(* Logix 5000 project; controller batter_comorfords vendor 1 type 14 code 222 rev 33.11; software revision 33.00 *)

TASK MainTask (continuous, watchdog 500 ms) : MainProgram
TASK SafetyTask (periodic, rate 20 ms, priority 10, watchdog 20 ms, safety) : SafetyProgram

MODULES
   Local : vendor 1 type 14 code 222 (5069 0, rev 33.11)
      PF525_Stirrer : PowerFlex 525-EENET (Ethernet 192.168.2.13, rev 5.2, Output RPI 20 ms)   // 0.75KW
      PF525_FeedingPump_2 : PowerFlex 525-EENET (Ethernet 192.168.2.15, rev 5.2, Output RPI 20 ms)   // 0.75 kW
      PF525_FeedingPump_1 : PowerFlex 525-EENET (Ethernet 192.168.2.14, rev 5.2, Output RPI 20 ms)   // 0.75 KW
      Manifold_with_color : 2198-H008-ERS2 (Ethernet 192.168.2.17, rev 7.1, DSafety_Input RPI 10 ms, CSafety_Output RPI 20 ms, AMotionDiagnostics RPI 1 ms)
      Manifold_without_color : 2198-H008-ERS2 (Ethernet 192.168.2.18, rev 7.1, AMotionDiagnostics RPI 1 ms, DSafety_Input RPI 10 ms, CSafety_Output RPI 20 ms)
      X_axis : 2198-H008-ERS2 (Ethernet 192.168.2.19, rev 7.1, AMotionDiagnostics RPI 1 ms, CSafety_Output RPI 20 ms, DSafety_Input RPI 10 ms)
      Y_axis : 2198-H008-ERS2 (Ethernet 192.168.2.20, rev 7.1, AMotionDiagnostics RPI 1 ms, CSafety_Output RPI 20 ms, DSafety_Input RPI 10 ms)
      Z_axis : 2198-H008-ERS2 (Ethernet 192.168.2.21, rev 7.1, AMotionDiagnostics RPI 1 ms, CSafety_Output RPI 20 ms, DSafety_Input RPI 10 ms)
      U1_MCC1_IO : 1734-AENTR (Ethernet 192.168.2.12, rev 6.1, Output RPI 20 ms)
         U1_MCC1_DIG_In_1 : 1734-IB8 (PointIO 3, rev 3.1)
         U1_MCC1_DIG_In_2 : 1734-IB8 (PointIO 4, rev 3.1)
         U1_MCC1_DIG_In_3 : 1734-IB8 (PointIO 5, rev 3.1)
         U1_MCC1_ANA_In_1 : vendor 1 type 115 code 210 (PointIO 6, rev 3.1, Input RPI 80 ms)
         U1_MCC1_DIG_Out_1 : vendor 1 type 7 code 231 (PointIO 7, rev 3.1)
         U1_MCC1_DIG_Out_2 : 1734-OB8 (PointIO 8, rev 3.1)
         U1_MCC1_DIG_Out_3 : 1734-OB8 (PointIO 9, rev 3.1)
         U1_MCC1_DIG_Out_4 : 1734-OB8 (PointIO 10, rev 3.1)
         U1_MCC1_ANA_Out_1 : 1734-OE2C (PointIO 11, rev 3.1, Output RPI 80 ms)
         U1_MCC1_Safety_DIG_In_1 : vendor 1 type 35 code 15 (PointIO 1, rev 2.1, Input RPI 10 ms, Output RPI 20 ms)
         U1_MCC1_Safety_DIG_Out_1 : vendor 1 type 35 code 16 (PointIO 2, rev 2.1, Input RPI 10 ms, Output RPI 20 ms)
      U4_MCC1_IO : 1734-AENTR (Ethernet 192.168.2.16, rev 6.1, Output RPI 20 ms)
         U4_MCC1_DIG_In_1 : 1734-IB8 (PointIO 3, rev 3.1)
         U4_MCC1_DIG_In_2 : 1734-IB8 (PointIO 4, rev 3.1)
         U4_MCC1_DIG_In_3 : 1734-IB8 (PointIO 5, rev 3.1)
         U4_MCC1_ANA_In_1 : 1734-IE4C (PointIO 6, rev 3.1, Input RPI 80 ms)
         U4_MCC1_ANA_In_2 : 1734-IE4C (PointIO 7, rev 3.1, Input RPI 80 ms)
         U4_MCC1_DIG_Out_1 : vendor 1 type 7 code 231 (PointIO 8, rev 3.1)
         U4_MCC1_DIG_Out_2 : vendor 1 type 7 code 231 (PointIO 9, rev 3.1)
         U4_MCC1_DIG_Out_3 : vendor 1 type 7 code 231 (PointIO 10, rev 3.1)
         U4_MCC1_ANA_Out_1 : 1734-OE2C (PointIO 11, rev 3.1, Output RPI 80 ms)
         U4_MCC1_Safety_DIG_In_1 : vendor 1 type 35 code 15 (PointIO 1, rev 2.1, Input RPI 10 ms, Output RPI 20 ms)
         U4_MCC1_Safety_DIG_Out_1 : vendor 1 type 35 code 16 (PointIO 2, rev 2.1, Input RPI 10 ms, Output RPI 20 ms)
END_MODULES

VAR_GLOBAL   (* controller tags *)
   IA_1_1_LT01 : ALIAS FOR U1_MCC1_IO:6:I.Ch0Data;   // Level buffertank
   IA_1_1_PT01 : ALIAS FOR U1_MCC1_IO:6:I.Ch1Data;   // Pressure feeding pump 1
   IA_1_2_LT01 : ALIAS FOR U1_MCC1_IO:6:I.Ch3Data;   // Level buffertank
   IA_1_2_PT01 : ALIAS FOR U1_MCC1_IO:6:I.Ch2Data;   // Pressure color injection
   IA_4_1_PT01 : ALIAS FOR U4_MCC1_IO:6:I.Ch1Data;   // Pressure manifold color
   IA_4_1_PT02 : ALIAS FOR U4_MCC1_IO:6:I.Ch3Data;   // Pressure manifold no color
   IA_4_1_TT01 : ALIAS FOR U4_MCC1_IO:6:I.Ch0Data;   // Temperature manifold color
   IA_4_1_TT02 : ALIAS FOR U4_MCC1_IO:6:I.Ch2Data;   // Temperature manifold no color
   ID_1_1_CIP_FAULT : ALIAS FOR U1_MCC1_IO:4:I.5;   // Fault CIP pump soft starter
   ID_1_1_GS01_1 : ALIAS FOR U1_MCC1_IO:3:I.5;   // Guard switch 1.1
   ID_1_1_GS01_2 : ALIAS FOR U1_MCC1_IO:3:I.6;   // Guard switch 1.2
   ID_1_1_GS01_3 : ALIAS FOR U1_MCC1_IO:3:I.7;   // Guard switch 1.3
   ID_1_1_LS01 : ALIAS FOR U1_MCC1_IO:4:I.1;   // Level switch feeding pump 1
   ID_1_1_OL_CIP : ALIAS FOR U1_MCC1_IO:4:I.4;   // Thermal overload CIP pump
   ID_1_1_OL_FAN : ALIAS FOR U1_MCC1_IO:3:I.0;   // Thermal overload Fan / Service socket
   ID_1_1_OL_M01 : ALIAS FOR U1_MCC1_IO:3:I.4;   // Thermal overload strirrer
   ID_1_1_OL_M02 : ALIAS FOR U1_MCC1_IO:4:I.0;   // Thermal overload feeding pump 1
   ID_1_1_OL_M03 : ALIAS FOR U1_MCC1_IO:4:I.2;   // Thermal overload feeding pump 2
   ID_1_1_PS01 : ALIAS FOR U1_MCC1_IO:3:I.1;   // Air pressure available
   ID_1_2_OL_M01 : ALIAS FOR U1_MCC1_IO:4:I.3;   // Thermal overload Color pump
   ID_4_1_GS01_1 : ALIAS FOR U4_MCC1_IO:4:I.0;   // Guard switch 1.1
   ID_4_1_GS01_2 : ALIAS FOR U4_MCC1_IO:4:I.1;   // Guard switch 1.2
   ID_4_1_GS01_3 : ALIAS FOR U4_MCC1_IO:4:I.2;   // Guard switch 1.3
   ID_4_1_GS02_1 : ALIAS FOR U4_MCC1_IO:4:I.3;   // Guard switch 2.1
   ID_4_1_GS02_2 : ALIAS FOR U4_MCC1_IO:4:I.4;   // Guard switch 2.2
   ID_4_1_GS02_3 : ALIAS FOR U4_MCC1_IO:4:I.5;   // Guard switch 2.3
   ID_4_1_GS03_1 : ALIAS FOR U4_MCC1_IO:5:I.0;   // Guard switch 3.1
   ID_4_1_GS03_2 : ALIAS FOR U4_MCC1_IO:5:I.1;   // Guard switch 3.2
   ID_4_1_GS03_3 : ALIAS FOR U4_MCC1_IO:5:I.2;   // Guard switch 3.3
   ID_4_1_GS04_1 : ALIAS FOR U4_MCC1_IO:5:I.3;   // Guard switch 4.1
   ID_4_1_GS04_2 : ALIAS FOR U4_MCC1_IO:5:I.4;   // Guard switch 4.2
   ID_4_1_GS04_3 : ALIAS FOR U4_MCC1_IO:5:I.5;   // Guard switch 4.3
   ID_4_1_OL_FAN : ALIAS FOR U4_MCC1_IO:3:I.0;   // Thermal overload Fan / Service socket
   ID_4_1_OL_M01 : ALIAS FOR U4_MCC1_IO:3:I.4;   // Thermal overload Power servo's
   ID_4_1_PS01 : ALIAS FOR U4_MCC1_IO:3:I.1;   // Air pressure available
   OA_1_2_M01 : ALIAS FOR U1_MCC1_IO:11:O.Ch0Data;   // Setpoint color pump
   OA_4_1_CV01 : ALIAS FOR U4_MCC1_IO:11:O.Ch0Data;   // Pressure valve manifold color
   OA_4_1_CV02 : ALIAS FOR U4_MCC1_IO:11:O.Ch1Data;   // Pressure valve manifold no color
   OD_1_1_CIP_START : ALIAS FOR U1_MCC1_IO:8:O.2;   // Start CIP pump soft starter
   OD_1_1_CIP_STOP : ALIAS FOR U1_MCC1_IO:8:O.3;   // Stop CIP pump soft starter
   OD_1_1_CV01 : ALIAS FOR U1_MCC1_IO:9:O.0;   // Valve spare
   OD_1_1_CV02 : ALIAS FOR U1_MCC1_IO:9:O.1;   // Valve drain after tank
   OD_1_1_CV03 : ALIAS FOR U1_MCC1_IO:9:O.2;   // Valve before CIP
   OD_1_1_CV04 : ALIAS FOR U1_MCC1_IO:9:O.3;   // Valve after CIP to pump 1
   OD_1_1_CV05 : ALIAS FOR U1_MCC1_IO:9:O.4;   // Valve after CIP to pump 2
   OD_1_1_CV06 : ALIAS FOR U1_MCC1_IO:9:O.5;   // Valve before feeding pump 1
   OD_1_1_CV07 : ALIAS FOR U1_MCC1_IO:9:O.6;   // Valve before feeding pump 2
   OD_1_1_CV08 : ALIAS FOR U1_MCC1_IO:9:O.7;   // Valve drain feeding pump 1
   OD_1_1_CV09 : ALIAS FOR U1_MCC1_IO:10:O.0;   // Valve drain feeding pump 2
   OD_1_1_CV10 : ALIAS FOR U1_MCC1_IO:10:O.1;   // Valve drain manifold
   OD_1_1_CV11 : ALIAS FOR U1_MCC1_IO:10:O.2;   // Valve drain before tank
   OD_1_1_CV12 : ALIAS FOR U1_MCC1_IO:10:O.3;   // Valve before sprinkler
   OD_1_1_CV13 : ALIAS FOR U1_MCC1_IO:10:O.4;   // Valve return tank
   OD_1_1_CV14 : ALIAS FOR U1_MCC1_IO:10:O.5;   // Valve hot water inlet
   OD_1_1_CV15 : ALIAS FOR U1_MCC1_IO:10:O.6;   // Valve cold water inlet
   OD_1_1_CV16 : ALIAS FOR U1_MCC1_IO:10:O.7;   // Valve spare
   OD_1_1_GS01 : ALIAS FOR U1_MCC1_IO:8:O.0;   // Guard switch 1 lock
   OD_1_1_SLBZ : ALIAS FOR U1_MCC1_IO:7:O.3;   // Signal column BUZZER
   OD_1_1_SLGN : ALIAS FOR U1_MCC1_IO:7:O.0;   // Signal column GN
   OD_1_1_SLRD : ALIAS FOR U1_MCC1_IO:7:O.2;   // Signal column RD
   OD_1_1_SLYE : ALIAS FOR U1_MCC1_IO:7:O.1;   // Signal column YE
   OD_1_2_M01 : ALIAS FOR U1_MCC1_IO:8:O.1;   // Enable color pump
   OD_4_1_CV01 : ALIAS FOR U4_MCC1_IO:10:O.0;   // Valve before manifold color
   OD_4_1_CV02 : ALIAS FOR U4_MCC1_IO:10:O.1;   // Valve before manifold no color
   OD_4_1_GS01 : ALIAS FOR U4_MCC1_IO:9:O.0;   // Guard switch 1 lock
   OD_4_1_GS02 : ALIAS FOR U4_MCC1_IO:9:O.1;   // Guard switch 2 lock
   OD_4_1_GS03 : ALIAS FOR U4_MCC1_IO:9:O.2;   // Guard switch 3 lock
   OD_4_1_GS04 : ALIAS FOR U4_MCC1_IO:9:O.3;   // Guard switch 4 lock
   OD_4_1_SLBZ : ALIAS FOR U4_MCC1_IO:8:O.3;   // Signal column BUZZER
   OD_4_1_SLGN : ALIAS FOR U4_MCC1_IO:8:O.0;   // Signal column GN
   OD_4_1_SLRD : ALIAS FOR U4_MCC1_IO:8:O.2;   // Signal column RD
   OD_4_1_SLYE : ALIAS FOR U4_MCC1_IO:8:O.1;   // Signal column YE
END_VAR

PROGRAM MainProgram   (* main routine MainRoutine *)

ROUTINE MainRoutine   (* ladder *)
END_ROUTINE
END_PROGRAM

PROGRAM SafetyProgram   (* main routine MainRoutine, safety *)

ROUTINE MainRoutine   (* ladder *)
END_ROUTINE
END_PROGRAM
